{attribute 'Tc2GvlVarNames'}
{attribute 'strict'}
{attribute 'to_String'}

TYPE Enum_Alarm_Others :
(
			Stn01ProcessTankHighTempAlarm								:= 300,
			Stn02ProcessTankHighTempAlarm                               := 301,
			Stn03ProcessTankHighTempAlarm                               := 302,
			Stn04ProcessTankHighTempAlarm                               := 303,
			Stn05ProcessTankHighTempAlarm                               := 304,
			Stn06ProcessTankHighTempAlarm                               := 305,
			Stn07ProcessTankHighTempAlarm                               := 306,
			Stn08ProcessTankHighTempAlarm                               := 307,
			Stn09ProcessTankHighTempAlarm                               := 308,
			Stn10ProcessTankHighTempAlarm                               := 309,
			ProcessTank1TempPreparationNoReadyAlarm                     := 315,
			ProcessTank2TempPreparationNoReadyAlarm                     := 316,
			ProcessTank3TempPreparationNoReadyAlarm                     := 317,
			ProcessTank4TempPreparationNoReadyAlarm                     := 318,
			ProcessTank5TempPreparationNoReadyAlarm                     := 319,
			ProcessTank6TempPreparationNoReadyAlarm                     := 320,
			ProcessTank7TempPreparationNoReadyAlarm                     := 321,
			ProcessTank8TempPreparationNoReadyAlarm                     := 322,
			ProcessTank9TempPreparationNoReadyAlarm                     := 323,
			ProcessTank1TempOver1StLimitAlarm                           := 330,
			ProcessTank2TempOver1StLimitAlarm                           := 331,
			ProcessTank3TempOver1StLimitAlarm                           := 332,
			ProcessTank4TempOver1StLimitAlarm                           := 333,
			ProcessTank5TempOver1StLimitAlarm                           := 334,
			ProcessTank6TempOver1StLimitAlarm                           := 335,
			ProcessTank7TempOver1StLimitAlarm                           := 336,
			ProcessTank8TempOver1StLimitAlarm                           := 337,
			ProcessTank9TempOver1StLimitAlarm                           := 338,
			ProcessTank10TempOver1StLimitAlarm                          := 339,
			ProcessTank1TempOver2NdLimitAlarm                           := 346,
			ProcessTank2TempOver2NdLimitAlarm                           := 347,
			ProcessTank3TempOver2NdLimitAlarm                           := 348,
			ProcessTank4TempOver2NdLimitAlarm                           := 349,
			ProcessTank5TempOver2NdLimitAlarm                           := 350,
			ProcessTank6TempOver2NdLimitAlarm                           := 351,
			ProcessTank7TempOver2NdLimitAlarm                           := 352,
			ProcessTank8TempOver2NdLimitAlarm                           := 353,
			ProcessTank9TempOver2NdLimitAlarm                           := 354,
			ProcessTank10TempOver2NdLimitAlarm                          := 355,
			ProcessTank11TempOver2NdLimitAlarm                          := 356,
			ProcessTank12TempOver2NdLimitAlarm                          := 357,
			IncTempOver2NdLimitAlarm                                    := 358,
			StnWaterJacketTempOver2NdLimitAlarm                         := 359,
			ProcessTank1ConductivityLowAlarm                            := 360,
			ProcessTank2ConductivityLowAlarm                            := 361,
			ProcessTank3ConductivityLowAlarm                            := 362,
			ProcessTank4ConductivityLowAlarm                            := 363,
			ProcessTank5ConductivityLowAlarm                            := 364,
			ProcessTank6ConductivityLowAlarm                            := 365,
			ProcessTank7ConductivityLowAlarm                            := 366,
			ProcessTank8ConductivityLowAlarm                            := 367,
			ProcessTank1PressureSwitchLowAlarm                          := 368,
			ProcessTank2PressureSwitchLowAlarm                          := 369,
			ProcessTank3PressureSwitchLowAlarm                          := 370,
			ProcessTank4PressureSwitchLowAlarm                          := 371,
			ProcessTank5PressureSwitchLowAlarm                          := 372,
			ProcessTank6PressureSwitchLowAlarm                          := 373,
			ProcessTank7PressureSwitchLowAlarm                          := 374,
			ProcessTank8PressureSwitchLowAlarm                          := 375,
			ProcessTank9PressureSwitchLowAlarm                          := 376,
			ProcessTank1ConductivityHighAlarm                           := 380,
			ProcessTank2ConductivityHighAlarm                           := 381,
			ProcessTank3ConductivityHighAlarm                           := 382,
			ProcessTank4ConductivityHighAlarm                           := 383,
			ProcessTank5ConductivityHighAlarm                           := 384,
			ProcessTank6ConductivityHighAlarm                           := 385,
			ProcessTank7ConductivityHighAlarm                           := 386,
			ProcessTank8ConductivityHighAlarm                           := 387,
			ProcessTank1PressureSwitchHighAlarm                         := 388,
			ProcessTank2PressureSwitchHighAlarm                         := 389,
			ProcessTank3PressureSwitchHighAlarm                         := 390,
			ProcessTank4PressureSwitchHighAlarm                         := 391,
			ProcessTank5PressureSwitchHighAlarm                         := 392,
			ProcessTank6PressureSwitchHighAlarm                         := 393,
			ProcessTank7PressureSwitchHighAlarm                         := 394,
			ProcessTank8PressureSwitchHighAlarm                         := 395,
			ProcessTank9PressureSwitchHighAlarm                         := 396,
			ProcessTank1BadBasket_OverToleranceTime                     := 400,
			ProcessTank2BadBasket_OverToleranceTime                     := 401,
			ProcessTank3BadBasket_OverToleranceTime                     := 402,
			ProcessTank4BadBasket_OverToleranceTime                     := 403,
			ProcessTank5BadBasket_OverToleranceTime                     := 404,
			ProcessTank6BadBasket_OverToleranceTime                     := 405,
			ProcessTank7BadBasket_OverToleranceTime                     := 406,
			ProcessTank8BadBasket_OverToleranceTime                     := 407,
			ProcessTank9BadBasket_OverToleranceTime                     := 408,
			ProcessTank10BadBasket_OverToleranceTime                    := 409,
			ProcessTank11BadBasket_OverToleranceTime                    := 410,
			ProcessTank12BadBasket_OverToleranceTime                    := 411,
			Arm1OvertimeError                                           := 412,
			Arm2OvertimeError                                           := 413,
			SlowpullLifterError                                         := 414,
			ProcessTank1DosingPumpHealthACheckPulseError                := 415,
			ProcessTank2DosingPumpHealthACheckPulseError                := 416,
			ProcessTank3DosingPumpHealthACheckPulseError                := 417,
			ProcessTank4DosingPumpHealthACheckPulseError				:= 418,
			Arm1VerticalUpOverTravelAlarm                               := 421,
			Arm1VerticalDownOverTravelAlarm                             := 422,
			Arm1VerticalErrorStopAlarm                                  := 423,
			Arm1HorizontalLoadingOverTravelAlarm                        := 424,
			Arm1HorizontalUnloadingOverTravelAlarm                      := 425,
			Arm1HorizontalErrorStopAlarm                                := 426,
			SlowpullUpOverTravelAlarm                                   := 427,
			SlowpullDownOverTravelAlarm                                 := 428,
			SlowpullErrorStopAlarm                                      := 429,
			DcPowerUnknownStatusAlarm                                   := 430,
			UpsCommUnknownStatusAlarm                                   := 431,
			BatteryReplacementRequestAlarm                              := 432,
			UpsCommErrorAlarm                                           := 433,
			Arm1VerticalAxisError                                       := 434,
			Arm1HorizontalAxisError                                     := 435,
			Arm2VerticalAxisError                                       := 436,
			Arm2HorizontalAxisError                                     := 437,
			MasterTimeBlockWriteArmDataError                            := 438,
			MasterTimeBlockWriteStnDataError                            := 439,
			MasterTimeBlockNoAvailableSlotError                         := 440,
			VacuumPumpRoutineServiceReminderAlarmReached				:= 441,
			VacuumPumpMajorWarningServiceReminder						:= 442,
			VacuumPumpMajorServiceReminderAlarmReached					:= 443,	
			LoadingCallArmSpeedProfileMemoryError                       := 444,
			LoadingCallPickStationNoError                               := 445,
			LoadingCallTransferStationNoError                           := 446,
			LoadingCallUpDownPatternMemoryError                         := 447,
			LoadingInvalidProductRecipeNoErrorHold                      := 448,
			LoadingInvalidProductRecipeStepErrorHold                    := 449,
			StationCallArmSpeedProfileMemoryError                       := 450,
			StationCallPickStationNoError                               := 451,
			StationCallTransferStationNoError                           := 452,
			StationCallUpDownPatternMemoryError                         := 453,
			StationInvalidProductRecipeNoErrorHold                      := 454,
			StationInvalidProductRecipeStepErrorHold                    := 455

);
END_TYPE

(* stored: Version 1.1.0.1, ProductVersion 3.1.4024.12
   DUT Enum_Alarm_Others: Id {86d6ef8f-c081-4000-82d7-b72a39d8337b} *)
